// TIA Portal V20 export
TYPE "typeUnitCommunicationControlNodeConveyorA"
// stored: Namespace Unit1.Em13
   STRUCT
      noInterference { ExternalWritable := 'False'} : Bool;
      requestPart { ExternalWritable := 'False'} : Bool;
      qrReadComplete { ExternalWritable := 'False'} : Bool;
      ungripRequest { ExternalWritable := 'False'} : Bool;
      loadComplete { ExternalWritable := 'False'} : Bool;
   END_STRUCT;
END_TYPE
